ABB RobotStudio station: Solution_1.rspag

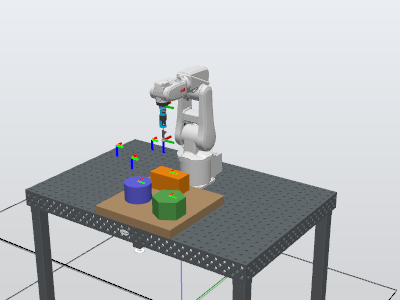
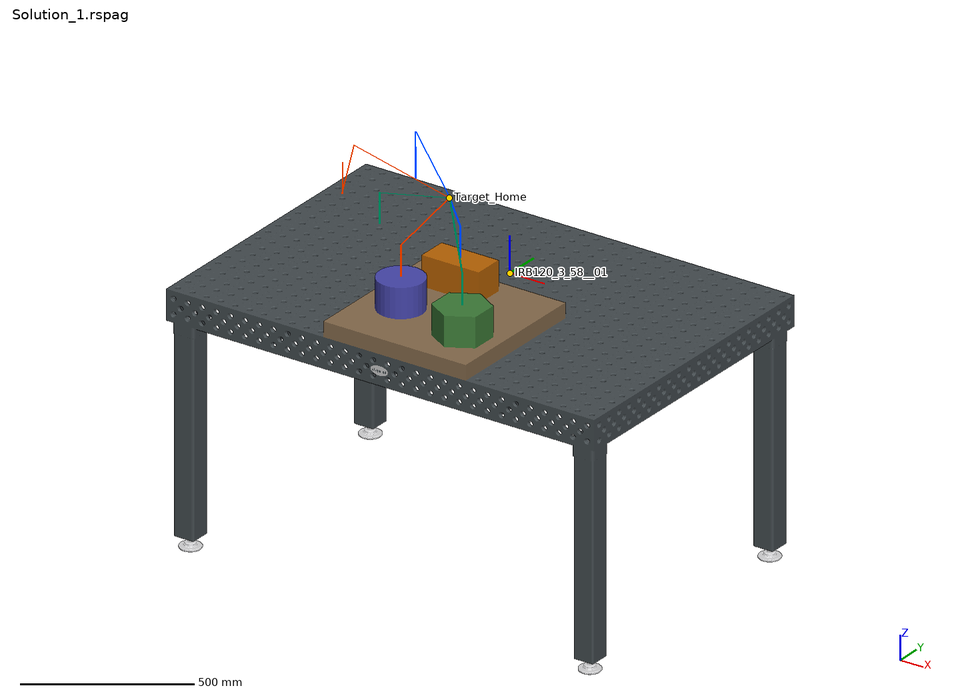
[picture v1: parts stored in the station drawn from their meshes, with robot base, taught points and paths (robot models come from the ABB library and are not in the file)]
--- station ---
Station Solution_1_Template_1 (saved by RobotStudio 22.3.10190.2)
Controller Controller1, task T_ROB1: task frame (RAPID world) sits at (0, 150, 830) mm, rotated rx 0 ry 0 rz -90 deg in the station
Controller Controller1
  mechanical unit ROB_1: IRB120_3_58__01, 6 joints, base frame (0, 0, 0) mm
Layout (positions relative to the parent item):
  - table [part] at (-200, -500, 830) mm, size 500 x 500 x 50 mm
  - object_1 [part] at (-200, -500, 830) mm, size 200 x 100 x 150 mm
  - object_2 [part] at (-200, -500, 830) mm, size 149.5 x 149.7 x 150 mm
  - object_3 [part] at (-200, -500, 830) mm, size 155.5 x 179.5 x 150 mm
  - siegmund_1500_1000 [part], size 1500 x 1010.3 x 830 mm
  - object_11 [part] at (-200, -500, 830) mm, size 200 x 100 x 150 mm
  - object_22 [part] at (-200, -500, 830) mm, size 149.5 x 149.7 x 150 mm
  - object_33 [part] at (-200, -500, 830) mm, size 155.5 x 179.5 x 150 mm
  - IRB120_3_58__01 [mechanism, from Robots\IRB120_3_58_G_01.rslib] at (0, 150, 830) mm, rotated rx 0 ry 0 rz -90 deg; joint values [0, 0, 0, 0, 1.5708, 0] (rad or m)
  - smc_gripper [mechanism, from Libraries\smc_gripper.rslib] at (0, -152, 1388) mm, rotated rx 180 ry 0 rz 90 deg
  - Positioner [smart component, from Components\Positioner.rslib]
      properties: Object=object_1; Position=[-0.6 -0.15 0.83]; Orientation=[0 0 0]; Reference=Global; ReferenceObject=(none)
  - Attacher [smart component, from Components\Attacher.rslib]
      properties: Parent=smc_gripper; Flange=0; Child=object_1; Mount=false; Offset=[0 0 0]; Orientation=[0 0 0]
  - Detacher [smart component, from Components\Detacher.rslib]
      properties: Child=object_1; KeepPosition=true
  - Positioner_2 [smart component, from Components\Positioner.rslib]
      properties: Object=object_2; Position=[-0.65 -0.15 0.83]; Orientation=[0 0 0]; Reference=Global; ReferenceObject=(none)
  - Positioner_3 [smart component, from Components\Positioner.rslib]
      properties: Object=object_3; Position=[-0.7 -0.2 0.83]; Orientation=[0 0 0]; Reference=Global; ReferenceObject=(none)
  - Attacher_2 [smart component, from Components\Attacher.rslib]
      properties: Parent=smc_gripper; Flange=0; Child=object_2; Mount=false; Offset=[0 0 0]; Orientation=[0 0 0]
  - Detacher_2 [smart component, from Components\Detacher.rslib]
      properties: Child=object_2; KeepPosition=true
  - Attacher_3 [smart component, from Components\Attacher.rslib]
      properties: Parent=smc_gripper; Flange=0; Child=object_3; Mount=false; Offset=[0 0 0]; Orientation=[0 0 0]
  - Detacher_3 [smart component, from Components\Detacher.rslib]
      properties: Child=object_3; KeepPosition=true
Attachment: smc_gripper is attached to IRB120_3_58__01 / Link6
Collision set CollisionSet_1: object_1 against object_2, object_3, near miss 0 m
Collision set Kolizní Sada_1: object_2 against object_3, object_1, near miss 0 m
Collision set Kolizní Sada_2: object_3 against object_2, object_1, near miss 0 m
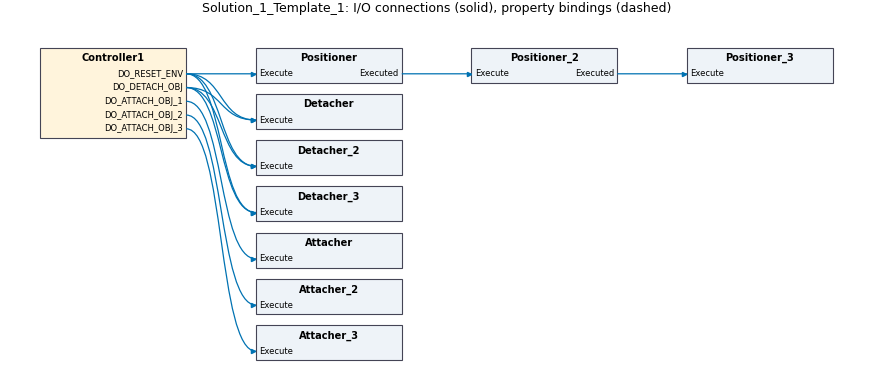
Station logic (signal -> signal, property => property):
  Controller1.DO_RESET_ENV -> Positioner.Execute
  Controller1.DO_DETACH_OBJ -> Detacher.Execute
  Positioner.Executed -> Positioner_2.Execute
  Positioner_2.Executed -> Positioner_3.Execute
  Controller1.DO_ATTACH_OBJ_1 -> Attacher.Execute
  Controller1.DO_ATTACH_OBJ_2 -> Attacher_2.Execute
  Controller1.DO_DETACH_OBJ -> Detacher_2.Execute
  Controller1.DO_DETACH_OBJ -> Detacher_3.Execute
  Controller1.DO_ATTACH_OBJ_3 -> Attacher_3.Execute
  Controller1.DO_RESET_ENV -> Detacher.Execute
  Controller1.DO_RESET_ENV -> Detacher_2.Execute
  Controller1.DO_RESET_ENV -> Detacher_3.Execute

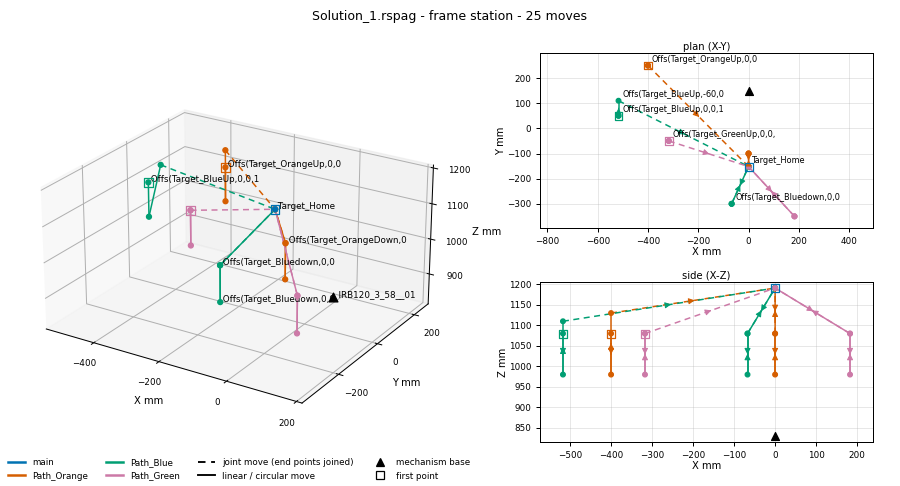
[picture p0: tool path of Solution_1.rspag in frame station, 25 of 25 moves have a stored position in this frame; points joined in program order, loops and branches not executed]
--- Backups/Controller1/RAPID/TASK1/PROGMOD/CalibData.mod ---
MODULE CalibData
    PERS tooldata smc_gripper:=[TRUE,[[0,0.004,197.001],[1,0,0,0]],[1,[0.207,-0.496,71.18],[1,0,0,0],0,0,0]];
ENDMODULE

--- Backups/Controller1/RAPID/TASK1/PROGMOD/Module1.mod ---
MODULE Module1
    CONST robtarget Target_Home:=[[302,0.004,360.999],[0,0,1,0],[0,0,0,0],[9E+09,9E+09,9E+09,9E+09,9E+09,9E+09]];
    CONST robtarget Target_OrangeUp:=[[-100,-400,150],[0,0,1,0],[-2,0,-2,0],[9E+09,9E+09,9E+09,9E+09,9E+09,9E+09]];
    CONST robtarget Target_OrangeDown:=[[250,0,150],[0,0,1,0],[-1,0,-1,0],[9E+09,9E+09,9E+09,9E+09,9E+09,9E+09]];
    CONST robtarget Target_BlueUp:=[[100,-517.298,150],[0,0,1,0],[-1,0,-1,0],[9E+09,9E+09,9E+09,9E+09,9E+09,9E+09]];
    CONST robtarget Target_BlueDown:=[[450,-67.298,150],[0,0,1,0],[-1,0,-1,0],[9E+09,9E+09,9E+09,9E+09,9E+09,9E+09]];
    CONST robtarget Target_GreenUp:=[[200,-317.298,150],[0,0,1,0],[-1,0,-1,0],[9E+09,9E+09,9E+09,9E+09,9E+09,9E+09]];
    CONST robtarget Target_GreenDown:=[[500,182.702,150],[0,0,1,0],[0,0,0,0],[9E+09,9E+09,9E+09,9E+09,9E+09,9E+09]];


    PROC main()
        ! Reset Env
        PulseDO DO_DETACH_OBJ;
        PulseDO DO_RESET_ENV;

        ! Home Position
        MoveJ Target_Home,v500,z50,smc_gripper\WObj:=wobj0;

        Path_Orange;

        Path_Blue;

        Path_Green;
    ENDPROC

    PROC Path_Orange()
        ! ORANGE OBJ
        MoveL Offs(Target_OrangeUp,0,0,100),v500,z50,smc_gripper\WObj:=wobj0;
        MoveL Offs(Target_OrangeUp,0,0,0),v500,fine,smc_gripper\WObj:=wobj0;

        PulseDO DO_ATTACH_OBJ_1;
        WaitTime 1.0;
        MoveL Offs(Target_OrangeUp,0,0,150),v500,z50,smc_gripper\WObj:=wobj0;

        ! Home Position
        MoveJ Target_Home,v500,z50,smc_gripper\WObj:=wobj0;

        MoveL Offs(Target_OrangeDown,0,0,100),v500,z50,smc_gripper\WObj:=wobj0;
        MoveL Offs(Target_OrangeDown,0,0,0),v500,fine,smc_gripper\WObj:=wobj0;

        PulseDO DO_DETACH_OBJ;
        WaitTime 1.0;
        MoveL Offs(Target_OrangeDown,0,0,100),v500,fine,smc_gripper\WObj:=wobj0;

        ! Home Position
        MoveJ Target_Home,v500,z50,smc_gripper\WObj:=wobj0;
    ENDPROC
    PROC Path_Blue()
        ! BLUE OBJ
        MoveL Offs(Target_BlueUp,0,0,100),v500,z50,smc_gripper\WObj:=wobj0;
        MoveL Offs(Target_BlueUp,0,0,0),v500,fine,smc_gripper\WObj:=wobj0;

        PulseDO DO_ATTACH_OBJ_2;
        WaitTime 1.0;
        MoveL Offs(Target_BlueUp,-60,0,130),v500,z50,smc_gripper\WObj:=wobj0;

        ! Home Position
        MoveJ Target_Home,v500,z50,smc_gripper\WObj:=wobj0;

        MoveL Offs(Target_Bluedown,0,0,100),v500,z50,smc_gripper\WObj:=wobj0;
        MoveL Offs(Target_Bluedown,0,0,0),v500,fine,smc_gripper\WObj:=wobj0;

        PulseDO DO_DETACH_OBJ;
        WaitTime 1.0;
        MoveL Offs(Target_Bluedown,0,0,100),v500,z50,smc_gripper\WObj:=wobj0;

        ! Home Position
        MoveJ Target_Home,v500,z50,smc_gripper\WObj:=wobj0;
    ENDPROC
    PROC Path_Green()
        ! GREEN OBJ
        MoveL Offs(Target_GreenUp,0,0,100),v500,z50,smc_gripper\WObj:=wobj0;
        MoveL Offs(Target_GreenUp,0,0,0),v500,fine,smc_gripper\WObj:=wobj0;

        PulseDO DO_ATTACH_OBJ_3;
        WaitTime 1.0;
        MoveL Offs(Target_GreenUp,0,0,100),v500,z50,smc_gripper\WObj:=wobj0;

        ! Home Position
        MoveJ Target_Home,v500,z50,smc_gripper\WObj:=wobj0;

        MoveL Offs(Target_GreenDown,0,0,100),v500,z50,smc_gripper\WObj:=wobj0;
        MoveL Offs(Target_GreenDown,0,0,0),v500,fine,smc_gripper\WObj:=wobj0;

        PulseDO DO_DETACH_OBJ;
        WaitTime 1.0;
        MoveL Offs(Target_GreenDown,0,0,100),v500,z50,smc_gripper\WObj:=wobj0;

        ! Home Position
        MoveJ Target_Home,v500,z50,smc_gripper\WObj:=wobj0;
    ENDPROC
ENDMODULE

--- Backups/Controller1/SYSPAR/EIO.cfg ---
EIO:CFG_1.0:6:1::
#
EIO_SIGNAL:

      -Name "DO_RESET_ENV" -SignalType "DO"

      -Name "DO_ATTACH_OBJ_1" -SignalType "DO"

      -Name "DO_DETACH_OBJ" -SignalType "DO"

      -Name "DO_ATTACH_OBJ_2" -SignalType "DO"

      -Name "DO_ATTACH_OBJ_3" -SignalType "DO"
